(* IEC 61131-3 sources: JaccoSigma/tempclass/Class/checkDirectory, 1 file *)

(* ---- checkDirectory.st ---- *)
(*!
<Class
	Name               = "checkDirectory"
	Revision           = "0.1"
	RealtimeTask       = "false"
	CyclicTask         = "false"
	BackgroundTask     = "false"
	DefBackground      = "100 ms"
	Sigmatek           = "false"
	OSInterface        = "false"
	HighPriority       = "false"
	Automatic          = "false"
	UpdateMode         = "Prescan"
	SharedCommandTable = "true"
	Objectsize         = "(638,120)">
	<Channels>
		<Server Name="ChangeDetected" Visualized="false" Initialize="false" WriteProtected="true" Retentive="false" Comment="Counts up every time something happens in the directory (member variable)"/>
		<Client Name="_MultiTask" Required="false" Internal="false"/>
		<Client Name="SigCLib" Required="false" Internal="false"/>
		<Client Name="SigCLib_or_Multitask" Required="false" Internal="false"/>
	</Channels>
	<RevDoku>
		<Owner Company="Sigmatek" Author="SchAnd"/>
		<Dokumentation Revision="0.1" Date="2021-07-02" Author="SchAnd" Company="Sigmatek" Description="Corrected way of x86 task creation, reworked dirscan to keep cpu load manageable&#13;&#10;Showcase will only detect changes within first 256 entries in directory though!"/>
	</RevDoku>
</Class>
*)
checkDirectory : CLASS
	TYPE
	  taskcreation :  //! <Type Public="true" Name="taskcreation"/>
	  (
	    sigcl_thread_create2:=1,
	    multitask_createthread:=2
	  )$UDINT;
	END_TYPE
  //Servers:
	ChangeDetected 	: SvrChCmd_DINT;
  //Clients:
	SigCLib 	: CltChCmd_SigCLib;
	_MultiTask 	: CltChCmd__MultiTask;
	SigCLib_or_Multitask 	: CltCh_taskcreation_PTofCls_checkDirectory;
  //Variables:
		checksum 	: UDINT;
		directory : ARRAY [0..255] OF CHAR;

		dirContent : ARRAY [0..255] OF _DDE_INFO;

		noelements 	: USINT;
		dirscan_ssw 	: DINT;
		searchhandle 	: DINT;
		currentelement : ARRAY [0..255] OF CHAR;

  //Functions:

	FUNCTION VIRTUAL GLOBAL Init;

	FUNCTION dirscan;

	FUNCTION __CDECL GLOBAL scanthread_SigCLib
		VAR_INPUT
			pThis 	: ^void;
		END_VAR
		VAR_OUTPUT
			continue (AL) 	: BOOL;
		END_VAR;

	FUNCTION __CDECL GLOBAL scanthread_MultiTask
		VAR_INPUT
			pThis 	: ^void;
		END_VAR;
  //Tables:
	FUNCTION @STD
		VAR_OUTPUT
			ret_code	: CONFSTATES;
		END_VAR;
	FUNCTION GLOBAL TAB @CT_;
END_CLASS;

#pragma usingLtd _MultiTask
#pragma usingLtd SigCLib

FUNCTION VIRTUAL GLOBAL checkDirectory::Init

  if _FirstScan then

    _strcpy(dest:=#directory[0], src:="c:\*");  // select a directory with < 256 elements inside

    if SigCLib_or_Multitask = sigcl_thread_create2 then  //Preferred
      sigclib_thread_create2(pfkt:=#scanthread_SigCLib(), priority:=8, time_us:=10000, pcookie:=this, name:="dirCheck_SigCLib");
    elsif SigCLib_or_Multitask = multitask_createthread then //Rather not use, stacksize unknown.
      _MultiTask.CREATETHREAD(taskfunction0:=#scanthread_MultiTask(), priority0:=8, stackSize0:=4kb, flags0:=0, parameter0:=this, name0:="dirCheck_MultiTask");
    end_if;

  end_if;

END_FUNCTION

FUNCTION checkDirectory::dirscan
  VAR
  	oldchks : udint;
  END_VAR

  case dirscan_ssw of
    0:
      noelements := 0;
      searchhandle := sigclib_findfirst(#directory[0], 0, 0, #dirContent[0], #currentelement[0], sizeof(currentelement));
      if searchhandle then
        dirscan_ssw += 1;
      end_if;
    1:
      if(currentelement[0] <> 0 & _strcmp(str1:=#currentelement[0], str2:=".") <> 0 & _strcmp(str1:=#currentelement[0], str2:="..") <> 0) then
        noelements += 1;
      end_if;
      if (sigclib_findnext(searchhandle, #dirContent[noelements], #currentelement[0], sizeof(currentelement)) <> 0 | noelements = 255) then //only check first 256 elements
        dirscan_ssw += 1;
      end_if;
    2:
      sigclib_findclose(searchhandle);
      searchhandle := 0;
      dirscan_ssw += 1;
    3:
      oldchks := checksum;
      checksum := sigclib_crc32(initval:=0, psrc:=#dirContent[0], length:=noelements*sizeof(_DDE_INFO));
      if checksum > 0 then
        dirscan_ssw := 0;
        if oldchks <> 0 & oldchks <> checksum then
          ChangeDetected += 1;
        end_if;
      end_if;

  end_case;

END_FUNCTION

FUNCTION __CDECL GLOBAL checkDirectory::scanthread_SigCLib
	VAR_INPUT
		pThis 	: ^void;
	END_VAR
	VAR_OUTPUT
		continue 	: BOOL;
	END_VAR

  this := pThis$^checkDirectory;
  dirscan();
  continue := true;

END_FUNCTION

FUNCTION __CDECL GLOBAL checkDirectory::scanthread_MultiTask
	VAR_INPUT
		pThis 	: ^void;
	END_VAR

  this := pThis$^checkDirectory;

  while 1 do

    dirscan();

    _MultiTask.TASKDELAY(timeout0:=10);

  end_while;

END_FUNCTION
